(* CODESYS project buffer_lib.library
   Company: Thomas More
   DefaultNamespace: Buffer
   Version: 1.0.0
   Placeholder: Buffer Lib
   Author: Arno Joosen
   Title: Buffer Lib

Project tree, tasks and I/O mapping:
  libraries: Tc2_Standard, * (Beckhoff Automation GmbH); Tc2_System, * (Beckhoff Automation GmbH); Tc3_Module, * (Beckhoff Automation GmbH)
  DUTs/
    data type Bool_ByteArray
    data type Buffer_Error
    data type Buffer_Layout
    data type Int_ByteArray
    data type Real_ByteArray
    data type String_ByteArray
  GVLs/
  POUs/
    Buffer_Layout_Configer/
      function Get_Layout_Size [ST]
      function Set_Buffer_Layout [ST]
    Read_Buffer/
      function Get_Bool_From_Buffer [ST]
      function Get_Int_From_Buffer [ST]
      function Get_Real_From_Buffer [ST]
      function Get_String_From_Buffer [ST]
    Wread_Buffer/
      function Set_Bool_Fom_Buffer [ST]
      function Set_Int_From_Buffer [ST]
      function Set_Real_From_Buffer [ST]
      function Set_String_From_Buffer [ST]
    program MAIN [ST]
  Version/
    global variables Global_Version
  VISUs/
*)

// DUTs/Bool_ByteArray
TYPE Bool_ByteArray :
UNION
	Value : BOOL;
	AValue:  BYTE;
END_UNION
END_TYPE

// DUTs/Buffer_Error
{attribute 'qualified_only'}
{attribute 'strict'}
TYPE Buffer_Error :
(
	None := 0,
	Overflow := 1,
	Array_Not_Enabelt := 2,
	Array_To_Small := 3,
	Layout_Not_Size_Buffer := 4,
	Read_Error := 5,
	Wread_Error := 6
) UINT;
END_TYPE

// DUTs/Buffer_Layout
TYPE Buffer_Layout :
STRUCT
	Buffer_Size : USINT := 64;
	
	// Bool
	Enabel_Bool_Array : BOOL := FALSE; // Bit in in-sight explorer
	Bool_Array_Offset : USINT := 0;
	Bool_Amount : USINT := 0;
	
	// Int
	Enabel_Int_Array : BOOL := TRUE; // int 16 bit in in-sight explorer
	Int_Array_Offset : USINT := 0;
	Int_Amount : USINT := 4;
	
	// Real
	Enabel_Real_Array : BOOL := TRUE; // float 32 bit in in-sight explorer
	Real_Array_Offset : USINT := 0;
	Real_Amount : USINT := 0;
	
	// String
	Enabel_String_Array : BOOL := FALSE; // string max 64 bytes in in-sight explorer
	String_Array_Offset : USINT := 0;
	String_Amount : USINT := 0;
	
END_STRUCT
END_TYPE

// DUTs/Int_ByteArray
TYPE Int_ByteArray :
UNION
	Value : INT;
	AValue:  ARRAY [0..1] OF BYTE;
END_UNION
END_TYPE

// DUTs/Real_ByteArray
TYPE Real_ByteArray :
UNION
	Value : REAL;
	AValue:  ARRAY [0..3] OF BYTE;
END_UNION
END_TYPE

// DUTs/String_ByteArray
TYPE String_ByteArray :
UNION
	Value : STRING[8];
	AValue:  ARRAY [0..8] OF BYTE;
END_UNION
END_TYPE

// Version/Global_Version
{attribute 'TcGenerated'}
{attribute 'no-analysis'}
{attribute 'linkalways'}
// This function has been automatically generated from the project information.
VAR_GLOBAL CONSTANT
	{attribute 'const_non_replaced'}
	stLibVersion_Buffer_Lib : ST_LibVersion := (iMajor := 1, iMinor := 0, iBuild := 0, iRevision := 0, nFlags := 0, sVersion := '1.0.0');
END_VAR

// POUs/Buffer_Layout_Configer/Get_Layout_Size
FUNCTION Get_Layout_Size : UINT
VAR_INPUT
	Layout : REFERENCE TO Buffer_Layout;
END_VAR
VAR
	Current_Buffer_Size : UINT := 0;
	i : UINT;
END_VAR

// calculate buffer size
// Bool array
IF Layout.Enabel_Bool_Array THEN 
	Current_Buffer_Size := Layout.Bool_Amount * 1; 
END_IF;
// Int array
IF Layout.Enabel_Int_Array THEN
	Current_Buffer_Size := Current_Buffer_Size + (Layout.Int_Amount * 2);
END_IF;
// Real array
IF Layout.Enabel_Real_Array THEN
	Current_Buffer_Size := Current_Buffer_Size + (Layout.Real_Amount * 4);
END_IF;
// String array
IF Layout.Enabel_String_Array THEN
	Current_Buffer_Size := Current_Buffer_Size + (Layout.String_Amount * 8);
END_IF;

Get_Layout_Size := Current_Buffer_Size;

END_FUNCTION

// POUs/Buffer_Layout_Configer/Set_Buffer_Layout
FUNCTION Set_Buffer_Layout : Buffer_Error
VAR_INPUT
	Buffer_Size : USINT;
	Bool_Amount : USINT;
	Int_Amount : USINT;
	Real_Amount : USINT;
	String_Amount : USINT;
END_VAR

VAR_IN_OUT
	Layout : Buffer_Layout;
END_VAR

VAR
	ClearLayout : Buffer_Layout;
	CurrentSize : USINT := 0;
END_VAR

Layout.Buffer_Size := Buffer_Size;

IF Bool_Amount > 0 THEN
	ClearLayout.Bool_Amount := Bool_Amount;
	ClearLayout.Bool_Array_Offset := CurrentSize;
	ClearLayout.Enabel_Bool_Array := TRUE;
	CurrentSize := CurrentSize + (Bool_Amount * 1);
ELSE
	ClearLayout.Enabel_Bool_Array := FALSE;
END_IF

IF Int_Amount > 0 THEN
	ClearLayout.Int_Amount := Int_Amount;
	ClearLayout.Int_Array_Offset := CurrentSize;
	ClearLayout.Enabel_Int_Array := TRUE;
	CurrentSize := CurrentSize + (Int_Amount * 2);
ELSE
	ClearLayout.Enabel_Int_Array := FALSE;
END_IF

IF Real_Amount > 0 THEN
	ClearLayout.Real_Amount := Real_Amount;
	ClearLayout.Real_Array_Offset := CurrentSize;
	Layout.Enabel_Real_Array := TRUE;
	CurrentSize := CurrentSize + (Real_Amount * 4);
ELSE
	Layout.Enabel_Real_Array := FALSE;
END_IF

IF String_Amount > 0 THEN
	ClearLayout.String_Amount := String_Amount;
	ClearLayout.String_Array_Offset := CurrentSize;
	ClearLayout.Enabel_String_Array := TRUE;
	CurrentSize := CurrentSize + (String_Amount * 9);
ELSE
	ClearLayout.Enabel_String_Array := FALSE;
END_IF

IF Layout.Buffer_Size < Get_Layout_Size(Layout:= ClearLayout) THEN
	Set_Buffer_Layout := Buffer_Error.Overflow;
ELSE
	Layout := ClearLayout;
	Set_Buffer_Layout := Buffer_Error.None;
END_IF

END_FUNCTION

// POUs/Read_Buffer/Get_Bool_From_Buffer
FUNCTION Get_Bool_From_Buffer : Buffer_Error
VAR_INPUT
	Num : USINT;
	Layout : REFERENCE TO Buffer_Layout;
END_VAR

VAR_IN_OUT
	Buffer : ARRAY [*] OF BYTE;
	Out : BOOL;
END_VAR

VAR
	Offset : USINT;
	CopyByte : BYTE;
	P_Int : POINTER TO BOOL;
	BufferSize : DINT;
	i : UINT;
END_VAR

BufferSize := UPPER_BOUND(Buffer, 1) - LOWER_BOUND(Buffer, 1); // berekent buffer size

IF BufferSize = Layout.Buffer_Size THEN
	Get_Bool_From_Buffer := Buffer_Error.Layout_Not_Size_Buffer; // return error dat buffer size niet overeen komt met buffer layout
	RETURN;
END_IF

IF NOT Layout.Enabel_Bool_Array THEN
	Get_Bool_From_Buffer := Buffer_Error.Array_Not_Enabelt; // return error data array niet enabelt is
	RETURN;
END_IF

IF Num > Layout.Bool_Amount THEN
	Get_Bool_From_Buffer := Buffer_Error.Array_To_Small; // return error data de num niet in de type array past
	RETURN;
END_IF

Offset := Layout.Bool_Array_Offset + (Num * 1);

IF Offset > BufferSize THEN // chek of float in buffer past met offset
	Out := FALSE; // return
	Get_Bool_From_Buffer := Buffer_Error.Read_Error; // return error read out of bouds van arry
	RETURN;
ELSE
	CopyByte := Buffer[Offset];
	P_Int := ADR(CopyByte); // maak een pinter van de buffer
	Get_Bool_From_Buffer := Buffer_Error.None;
	Out := P_Int^; // return
END_IF

END_FUNCTION

// POUs/Read_Buffer/Get_Int_From_Buffer
FUNCTION Get_Int_From_Buffer : Buffer_Error
VAR_INPUT
	Num : USINT;
	Layout : REFERENCE TO Buffer_Layout;
END_VAR

VAR_IN_OUT
	Buffer : ARRAY [*] OF BYTE;
	Out : INT;
END_VAR

VAR
	Offset : USINT;
	CopyArray : ARRAY [0..1] OF BYTE;
	P_Int : POINTER TO INT;
	BufferSize : DINT;
	i : UINT;
END_VAR

BufferSize := UPPER_BOUND(Buffer, 1) - LOWER_BOUND(Buffer, 1); // berekent buffer size

IF BufferSize = Layout.Buffer_Size THEN
	Get_Int_From_Buffer := Buffer_Error.Layout_Not_Size_Buffer; // return error dat buffer size niet overeen komt met buffer layout
	RETURN;
END_IF

IF NOT Layout.Enabel_Int_Array THEN
	Get_Int_From_Buffer := Buffer_Error.Array_Not_Enabelt; // return error data array niet enabelt is
	RETURN;
END_IF

IF Num > Layout.Int_Amount THEN
	Get_Int_From_Buffer := Buffer_Error.Array_To_Small; // return error data de num niet in de type array past
	RETURN;
END_IF

Offset := Layout.Int_Array_Offset + (Num * 2);

IF Offset + 2 > BufferSize THEN // chek of float in buffer past met offset
	Out := 0; // return
	Get_Int_From_Buffer := Buffer_Error.Read_Error; // return error read out of bouds van arry
	RETURN;
ELSE
	FOR i:=0 TO 1 BY 1 DO // copy data en swap naar een copy buffer
    	CopyArray[i] := Buffer[(1 - i) + Offset];
	END_FOR;
	P_Int := ADR(CopyArray); // maak een pinter van de buffer
	Get_Int_From_Buffer := Buffer_Error.None;
	Out := P_Int^; // return
END_IF

END_FUNCTION

// POUs/Read_Buffer/Get_Real_From_Buffer
FUNCTION Get_Real_From_Buffer : Buffer_Error
VAR_INPUT
	Num : USINT;
	Layout : REFERENCE TO Buffer_Layout;
END_VAR

VAR_IN_OUT
	Buffer : ARRAY [*] OF BYTE;
	Out : REAL;
END_VAR

VAR
	Offset : USINT;
	CopyArray : ARRAY [0..3] OF BYTE;
	P_Int : POINTER TO REAL;
	BufferSize : DINT;
	i : UINT;
END_VAR

BufferSize := UPPER_BOUND(Buffer, 1) - LOWER_BOUND(Buffer, 1); // berekent buffer size

IF BufferSize = Layout.Buffer_Size THEN
	Get_Real_From_Buffer := Buffer_Error.Layout_Not_Size_Buffer; // return error dat buffer size niet overeen komt met buffer layout
	RETURN;
END_IF

IF NOT Layout.Enabel_Real_Array THEN
	Get_Real_From_Buffer := Buffer_Error.Array_Not_Enabelt; // return error data array niet enabelt is
	RETURN;
END_IF

IF Num > Layout.Real_Amount THEN
	Get_Real_From_Buffer := Buffer_Error.Array_To_Small; // return error data de num niet in de type array past
	RETURN;
END_IF

Offset := Layout.Real_Array_Offset + (Num * 4);

IF Offset + 2 > BufferSize THEN // chek of float in buffer past met offset
	Out := 0;
	Get_Real_From_Buffer := Buffer_Error.Read_Error; // return error read out of bouds van arry
	RETURN;
ELSE
	FOR i:=0 TO 3 BY 1 DO // copy data en swap naar een copy buffer
    	CopyArray[i] := Buffer[(3 - i) + Offset];
	END_FOR;
	P_Int := ADR(CopyArray); // maak een pinter van de buffer
	Get_Int_From_Buffer := Buffer_Error.None;
	Out := P_Int^; // return
END_IF

END_FUNCTION

// POUs/Read_Buffer/Get_String_From_Buffer
FUNCTION Get_String_From_Buffer : Buffer_Error
VAR_INPUT
	Num : USINT;
	Layout : REFERENCE TO Buffer_Layout;
END_VAR

VAR_IN_OUT
	Buffer : ARRAY [*] OF BYTE;
	Out : STRING[8];
END_VAR

VAR
	Offset : USINT;
	CopyArray : ARRAY [0..7] OF BYTE;
	P_Int : POINTER TO STRING[8];
	BufferSize : DINT;
	i : UINT;
END_VAR

BufferSize := UPPER_BOUND(Buffer, 1) - LOWER_BOUND(Buffer, 1); // berekent buffer size

IF BufferSize = Layout.Buffer_Size THEN
	Get_Real_From_Buffer := Buffer_Error.Layout_Not_Size_Buffer; // return error dat buffer size niet overeen komt met buffer layout
	RETURN;
END_IF

IF NOT Layout.Enabel_Real_Array THEN
	Get_Real_From_Buffer := Buffer_Error.Array_Not_Enabelt; // return error data array niet enabelt is
	RETURN;
END_IF

IF Num > Layout.Real_Amount THEN
	Get_Real_From_Buffer := Buffer_Error.Array_To_Small; // return error data de num niet in de type array past
	RETURN;
END_IF

Offset := Layout.Real_Array_Offset + (Num * 9);

IF Offset + 8 > BufferSize THEN // chek of float in buffer past met offset
	Out := '';
	Get_Real_From_Buffer := Buffer_Error.Read_Error; // return error read out of bouds van arry
	RETURN;
ELSE
	FOR i:=0 TO 8 BY 1 DO // copy data en swap naar een copy buffer
    	CopyArray[i] := Buffer[(8 - i) + Offset];
	END_FOR;
	P_Int := ADR(CopyArray); // maak een pinter van de buffer
	Get_Int_From_Buffer := Buffer_Error.None;
	Out := P_Int^; // return
END_IF

END_FUNCTION

// POUs/Wread_Buffer/Set_Bool_Fom_Buffer
FUNCTION Set_Bool_Fom_Buffer : Buffer_Error
VAR_INPUT
	In : BOOL;
	Num : USINT;
	Layout : REFERENCE TO Buffer_Layout;
END_VAR

VAR_IN_OUT
	Buffer : ARRAY [*] OF BYTE;
END_VAR

VAR
	Offset : USINT;
	BufferSize : DINT;
	U_Int : Bool_ByteArray;
END_VAR

BufferSize := UPPER_BOUND(Buffer, 1) - LOWER_BOUND(Buffer, 1); // berekent buffer size

IF BufferSize = Layout.Buffer_Size THEN
	Set_Bool_Fom_Buffer := Buffer_Error.Layout_Not_Size_Buffer; // return error dat buffer size niet overeen komt met buffer layout
	RETURN;
END_IF

IF NOT Layout.Enabel_Bool_Array THEN
	Set_Bool_Fom_Buffer := Buffer_Error.Array_Not_Enabelt; // return error data array niet enabelt is
	RETURN;
END_IF

IF Num > Layout.Bool_Amount THEN
	Set_Bool_Fom_Buffer := Buffer_Error.Array_To_Small; // return error data de num niet in de type array past
	RETURN;
END_IF

Offset := Layout.Bool_Array_Offset + Num;

IF Offset > BufferSize THEN
	Set_Bool_Fom_Buffer := Buffer_Error.Wread_Error;
	RETURN;
ELSE
	U_Int.Value := In;
	Buffer[Offset] := U_Int.AValue;
	Set_Bool_Fom_Buffer := Buffer_Error.None;
END_IF

END_FUNCTION

// POUs/Wread_Buffer/Set_Int_From_Buffer
FUNCTION Set_Int_From_Buffer : Buffer_Error
VAR_INPUT
	In : INT;
	Num : USINT;
	Layout : REFERENCE TO Buffer_Layout;
END_VAR

VAR_IN_OUT
	Buffer : ARRAY [*] OF BYTE;
END_VAR

VAR
	Offset : USINT;
	BufferSize : DINT;
	U_Int : Int_ByteArray;
	i : UINT;
END_VAR

BufferSize := UPPER_BOUND(Buffer, 1) - LOWER_BOUND(Buffer, 1); // berekent buffer size

IF BufferSize = Layout.Buffer_Size THEN
	Set_Int_From_Buffer := Buffer_Error.Layout_Not_Size_Buffer; // return error dat buffer size niet overeen komt met buffer layout
	RETURN;
END_IF

IF NOT Layout.Enabel_Int_Array THEN
	Set_Int_From_Buffer := Buffer_Error.Array_Not_Enabelt; // return error data array niet enabelt is
	RETURN;
END_IF

IF Num > Layout.Int_Amount THEN
	Set_Int_From_Buffer := Buffer_Error.Array_To_Small; // return error data de num niet in de type array past
	RETURN;
END_IF

Offset := Layout.Int_Array_Offset + (Num * 2);

IF Offset + 1 > BufferSize THEN
	Set_Int_From_Buffer := Buffer_Error.Wread_Error;
	RETURN;
ELSE
	U_Int.Value := In;
	FOR i:=0 TO 1 BY 1 DO
		Buffer[Offset + i] := U_Int.AValue[i];
	END_FOR
	Set_Int_From_Buffer := Buffer_Error.None;
END_IF

END_FUNCTION

// POUs/Wread_Buffer/Set_Real_From_Buffer
FUNCTION Set_Real_From_Buffer : Buffer_Error
VAR_INPUT
	In : REAL;
	Num : USINT;
	Layout : REFERENCE TO Buffer_Layout;
END_VAR

VAR_IN_OUT
	Buffer : ARRAY [*] OF BYTE;
END_VAR

VAR
	Offset : USINT;
	BufferSize : DINT;
	U_Int : Real_ByteArray;
	i : UINT;
END_VAR

BufferSize := UPPER_BOUND(Buffer, 1) - LOWER_BOUND(Buffer, 1); // berekent buffer size

IF BufferSize = Layout.Buffer_Size THEN
	Set_Real_From_Buffer := Buffer_Error.Layout_Not_Size_Buffer; // return error dat buffer size niet overeen komt met buffer layout
	RETURN;
END_IF

IF NOT Layout.Enabel_Real_Array THEN
	Set_Real_From_Buffer := Buffer_Error.Array_Not_Enabelt; // return error data array niet enabelt is
	RETURN;
END_IF

IF Num > Layout.Real_Amount THEN
	Set_Real_From_Buffer := Buffer_Error.Array_To_Small; // return error data de num niet in de type array past
	RETURN;
END_IF

Offset := Layout.Real_Array_Offset + (Num * 4);

IF Offset + 3 > BufferSize THEN
	Set_Real_From_Buffer := Buffer_Error.Wread_Error;
	RETURN;
ELSE
	U_Int.Value := In;
	FOR i:=0 TO 3 BY 1 DO
		Buffer[Offset + i] := U_Int.AValue[i];
	END_FOR
	Set_Real_From_Buffer := Buffer_Error.None;
END_IF

END_FUNCTION

// POUs/Wread_Buffer/Set_String_From_Buffer
FUNCTION Set_String_From_Buffer : Buffer_Error
VAR_INPUT
	In : STRING;
	Num : USINT;
	Layout : REFERENCE TO Buffer_Layout;
END_VAR

VAR_IN_OUT
	Buffer : ARRAY [*] OF BYTE;
END_VAR

VAR
	Offset : USINT;
	BufferSize : DINT;
	CopyBuffer : String_ByteArray;
	i : UINT;
	EndTrigger : BOOL := FALSE;
END_VAR

BufferSize := UPPER_BOUND(Buffer, 1) - LOWER_BOUND(Buffer, 1); // berekent buffer size

IF BufferSize = Layout.Buffer_Size THEN
	Set_String_From_Buffer := Buffer_Error.Layout_Not_Size_Buffer; // return error dat buffer size niet overeen komt met buffer layout
	RETURN;
END_IF

IF NOT Layout.Enabel_String_Array THEN
	Set_String_From_Buffer := Buffer_Error.Array_Not_Enabelt; // return error data array niet enabelt is
	RETURN;
END_IF

IF Num > Layout.String_Amount THEN
	Set_String_From_Buffer := Buffer_Error.Array_To_Small; // return error data de num niet in de type array past
	RETURN;
END_IF

Offset := Layout.String_Array_Offset + (Num * 9);

IF Offset + 7 > BufferSize THEN
	Set_String_From_Buffer := Buffer_Error.Wread_Error;
	RETURN;
ELSE
	CopyBuffer.Value := In;
	FOR i:=0 TO 8 BY 1 DO
		IF (NOT (CopyBuffer.AValue[i] = 0)) AND (NOT EndTrigger) THEN
			Buffer[Offset + i] := CopyBuffer.AValue[i];
		ELSE
			EndTrigger := TRUE;
			Buffer[Offset + i] := 0;
		END_IF;
	END_FOR
	Set_String_From_Buffer := Buffer_Error.None;
END_IF

END_FUNCTION

// POUs/MAIN
PROGRAM MAIN
VAR
	fbGetCurTaskIdx  : GETCURTASKINDEX;
	
	Layout : Buffer_Layout;
	Buffer : ARRAY[0..63] OF BYTE;
	
	// out var
	VarEen : INT;
	VarTwee : INT;
END_VAR


Set_Buffer_Layout(
	Buffer_Size:= 64, 
	Bool_Amount:= 0, 
	Int_Amount:= 0, 
	Real_Amount:= 0, 
	String_Amount:= 2, 
	Layout:= Layout);

Set_Int_From_Buffer(
	In:= 300, 
	Num:= 0, 
	Layout:= Layout, 
	Buffer:= Buffer);
	
Set_Int_From_Buffer(
	In:= 30, 
	Num:= 1, 
	Layout:= Layout, 
	Buffer:= Buffer);
	
Set_Bool_Fom_Buffer(
	In:= TRUE, 
	Num:= 0, 
	Layout:= Layout, 
	Buffer:= Buffer);
	
	
Set_Bool_Fom_Buffer(
	In:= TRUE, 
	Num:= 1, 
	Layout:= Layout, 
	Buffer:= Buffer);
	
	
Set_Real_From_Buffer(
	In:= 3.55, 
	Num:= 0, 
	Layout:= Layout, 
	Buffer:= Buffer);
	
Set_Real_From_Buffer(
	In:= 10.66, 
	Num:= 1, 
	Layout:= Layout, 
	Buffer:= Buffer);
	
	
Set_String_From_Buffer(
	In:= 'AAAAA', 
	Num:= 0, 
	Layout:= Layout, 
	Buffer:= Buffer);
	
Set_String_From_Buffer(
	In:= 'AAAAAAAA', 
	Num:= 1, 
	Layout:= Layout, 
	Buffer:= Buffer);

END_PROGRAM
